PROGRAM MAIN
VAR
	timeElapsed : Counter;
	recordedTime : TIME ;
	valve : CloseValve;
	valveClose : BOOL ;
END_VAR


(* IF NOT GVL.sensorN1 AND readyToMeasureTime THEN
	startTime := TIME() ;
	measuringStarted := TRUE ;
END_IF 

IF NOT GVL.sensorN2 AND measuringStarted THEN
	stopTime := TIME() ;
END_IF *)

//startMeasurement := TRUE;


valve(closeValve => GVL.valveClose);

timeElapsed( timeElapsed => recordedTime);

END_PROGRAM

(* stored: Version 1.1.0.1, ProductVersion 3.1.4024.13
   POU MAIN: Id {26a15cae-5634-4149-81e6-7ccf156c7169}, SpecialFunc None *)
